DATA_BLOCK "hmiDB"
TITLE = hmiDB
{ S7_Optimized_Access := 'FALSE' }
AUTHOR : JB
VERSION : 0.1
NON_RETAIN
//Contains all the tags that a HMI will need to interact with, sorted in sections. Each cycle, the inputs are read, and the outputs are updated.
   STRUCT
      system : Struct
         general : Struct
            errorPLC { ExternalWritable := 'False'} : Bool;   // Shows error in the PLC
            requestClearFaults : Bool;   // Button input, to clear faults
            systemFault { ExternalWritable := 'False'} : Bool;   // Indicator, to show if fault is present
            faultCount { ExternalWritable := 'False'} : Int;   // Count of how many faults are present
            coolantStatus { ExternalWritable := 'False'} : Bool;   // Indicator, to show if coolant is active
            faultArray { ExternalWritable := 'False'} : Array[0..100] of Bool;
            messageBuffer { ExternalWritable := 'False'} : Array[0..29] of Int;
            bufferIndex { ExternalWritable := 'False'} : Int;
         END_STRUCT;
         ionSource : Struct
            general : Struct
               status : Int;   // Status, enabled=+1, fault=+2
               modeCurrent { ExternalWritable := 'False'} : Int;   // Display field showing source mode
               requestStart : Bool;   // Button input, to start the source
               requestStop : Bool;   // Button input, to stop the source
               requestCondition : Bool;   // Tickbox input
               conditioningPaused { ExternalWritable := 'False'} : Bool;   // Indicator, to show if conditioning has paused
               requestPause : Bool;   // Button input, to pause the source
               requestResume : Bool;   // Button input, to resume the source
               bodyTempC { ExternalWritable := 'False'} : Real;   // Display number, showing source temperature
               bodyTempOkay { ExternalWritable := 'False'} : Bool;   // Indicator, to show if source is cold enough - affects colour of above number
               beamVoltage { ExternalWritable := 'False'} : Real;
               doorStatus : Bool;
            END_STRUCT;
            ioniser : Struct
               status { ExternalWritable := 'False'} : Int;   // Status for ioniser, enabled=+1, fault=+2
               hmiSetpointWEnabled { ExternalWritable := 'False'} : Bool;   // Determines if power setpoint can be written too by HMI
               hmiSetpointWEntry : Real;   // Entry field, to set ioniser power
               hmiSetpointWEntryMin { ExternalWritable := 'False'} : Real;
               hmiSetpointWEntryMax { ExternalWritable := 'False'} : Real;
               readbackW { ExternalWritable := 'False'} : Real;   // Display field, showing ioniser power
               powerRatio : Real;
               filament : Struct
                  status : Int;   // Status, enabled=+1, fault=+2
                  readbackV : Real;
                  readbackA : Real;
                  readbackW : Real;
               END_STRUCT;
               thermionic : Struct
                  status : Int;   // Status, enabled=+1, fault=+2
                  readbackV : Real;
                  readbackA : Real;
                  readbackW : Real;
               END_STRUCT;
            END_STRUCT;
            target : Struct
               status { ExternalWritable := 'False'} : Int;   // Status for target, 0=off/disabled, 1=on/enabled, 2=fault
               hmiSetpointVEnabled { ExternalWritable := 'False'} : Bool;   // Determines if voltage setpoint can be written too by HMI
               hmiSetpointVEntry : Real;   // Entry field, to set target voltage
               hmiSetpointVEntryMin { ExternalWritable := 'False'} : Real;
               hmiSetpointVEntryMax { ExternalWritable := 'False'} : Real;
               readbackV { ExternalWritable := 'False'} : Real;   // Display field, showing target voltage
               readbackA { ExternalWritable := 'False'} : Real;   // Display field, showing target current
               readbackW { ExternalWritable := 'False'} : Real;   // Display field, showing target power
            END_STRUCT;
            extraction : Struct
               status { ExternalWritable := 'False'} : Int;   // Status for extraction, 0=off/disabled, 1=on/enabled, 2=fault
               hmiSetpointVEnabled { ExternalWritable := 'False'} : Bool;   // Determines if extraction setopint can be written too by HMI
               hmiSetpointVEntry : Real;   // Entry field, to set extraction voltage
               hmiSetpointVEntryMin { ExternalWritable := 'False'} : Real;
               hmiSetpointVEntryMax { ExternalWritable := 'False'} : Real;
               readbackV { ExternalWritable := 'False'} : Real;   // Display field, showing extraction voltage
               readbackA { ExternalWritable := 'False'} : Real;   // Display field, showing extraction current
               readbackW { ExternalWritable := 'False'} : Real;   // Display field, showing extraction power
            END_STRUCT;
            cesium : Struct
               status { ExternalWritable := 'False'} : Int;   // Status for cesium, 0=off/disabled, 1=on/enabled, 2=fault
               hmiSetpointCEnabled { ExternalWritable := 'False'} : Bool;   // Determines if temperature setpoint can be written too by HMI
               hmiSetpointCEntry : Real;   // Entry field, to set cesium temperature
               hmiSetpointCEntryMin { ExternalWritable := 'False'} : Real;
               hmiSetpointCEntryMax { ExternalWritable := 'False'} : Real;
               readbackC { ExternalWritable := 'False'} : Real;   // Display field, showing cesium temperature
               heaterOn { ExternalWritable := 'False'} : Bool;   // Indicator, to show if heat is being applied
               coolantOn { ExternalWritable := 'False'} : Bool;   // Indicator, to show if coolant is active
            END_STRUCT;
         END_STRUCT;
         vacuumSystem : Struct
            gauges : Struct
               source : Struct
                  readback_mB : Real;
                  status : Bool;
               END_STRUCT;
               beamline : Struct
                  readback_mB : Real;
                  status : Bool;
               END_STRUCT;
               chamber_UHV_gauge : Struct
                  readback_mB : Bool;
                  status : Bool;
               END_STRUCT;
               chamber_reg_gauge : Struct
                  readback_mB : Real;
                  status : Bool;
               END_STRUCT;
            END_STRUCT;
            pumps : Struct
               roughing { ExternalWritable := 'False'} : Struct
                  source { ExternalWritable := 'False'} : Struct
                     status { ExternalWritable := 'False'} : Bool;
                  END_STRUCT;
                  beamline { ExternalWritable := 'False'} : Struct
                     status { ExternalWritable := 'False'} : Bool;
                  END_STRUCT;
                  loadlock { ExternalWritable := 'False'} : Struct
                     status { ExternalWritable := 'False'} : Bool;
                  END_STRUCT;
               END_STRUCT;
               turbo { ExternalWritable := 'False'} : Struct
                  source_1 { ExternalWritable := 'False'} : Struct
                     status { ExternalWritable := 'False'} : Bool;
                     speed { ExternalWritable := 'False'} : Real;
                     on_hours { ExternalWritable := 'False'} : Real;
                  END_STRUCT;
                  source_2 { ExternalWritable := 'False'} : Struct
                     status { ExternalWritable := 'False'} : Bool;
                     speed { ExternalWritable := 'False'} : Real;
                     on_hours { ExternalWritable := 'False'} : Real;
                  END_STRUCT;
                  beamline { ExternalWritable := 'False'} : Struct
                     status { ExternalWritable := 'False'} : Bool;
                     speed { ExternalWritable := 'False'} : Real;
                     on_hours { ExternalWritable := 'False'} : Real;
                  END_STRUCT;
                  chamber { ExternalWritable := 'False'} : Struct
                     status { ExternalWritable := 'False'} : Bool;
                     speed { ExternalWritable := 'False'} : Real;
                     on_hours { ExternalWritable := 'False'} : Real;
                  END_STRUCT;
                  loadlock { ExternalWritable := 'False'} : Struct
                     status { ExternalWritable := 'False'} : Bool;
                     speed { ExternalWritable := 'False'} : Real;
                     on_hours { ExternalWritable := 'False'} : Real;
                  END_STRUCT;
               END_STRUCT;
               titanium : Struct
                  chamber_1 : Struct
                     on_time_s : Real;
                     off_time_s : Real;
                     nominal_current_A : Real;
                     filament_1 : Struct
                        status : Bool;
                        on_hours : Real;
                        cycles : Int;
                     END_STRUCT;
                  END_STRUCT;
               END_STRUCT;
               ion : Struct
                  chamber_1 : Struct
                     voltage_readback_V : Real;
                     current_readback_A : Real;
                     on_hours : Real;
                  END_STRUCT;
               END_STRUCT;
            END_STRUCT;
            valves : Struct
               gate : Struct
                  "source-beamline" : Struct
                     open : Bool;
                     cycles : Int;
                     requestOpen : Bool;
                  END_STRUCT;
                  "beamline-chamber" : Struct
                     open : Bool;
                     cycles : Int;
                     requestOpen : Bool;
                  END_STRUCT;
                  "chamber-loadlock" : Struct
                     open : Bool;
                     cycles : Int;
                  END_STRUCT;
               END_STRUCT;
               pneumatic : Struct
                  placeholder : Bool;
               END_STRUCT;
            END_STRUCT;
         END_STRUCT;
         beamline : Struct
            magnet : Struct
               status : Int;
               static_active : Bool;
               hmiSetpointAEnabled : Bool;
               hmiSetpointAEntry : Real;
               hmiSetpointAEntryMin : Real;
               hmiSetpointAEntryMax : Real;
               readbackV : Real;
               readbackA : Real;
               outputEnabled : Bool;
               fault : Bool;
            END_STRUCT;
            steerers : Struct
               x : Struct
                  status : Bool;
                  hmiSetpointVEnabled : Bool;
                  hmiSetpointVEntry : Real;
                  hmiSetpointVEntryMin : Real;
                  hmiSetpointVEntryMax : Real;
                  readbackV : Real;
                  readbackA : Real;
                  outputEnabled : Bool;
                  fault : Bool;
               END_STRUCT;
               y : Struct
                  status : Bool;
                  hmiSetpointVEnabled : Bool;
                  hmiSetpointVEntry : Real;
                  hmiSetpointVEntryMin : Real;
                  hmiSetpointVEntryMax : Real;
                  readbackV : Real;
                  readbackA : Real;
                  outputEnabled : Bool;
                  fault : Bool;
               END_STRUCT;
            END_STRUCT;
            einzels : Struct
               lens1 : Struct
                  status : Bool;
                  hmiSetpointVEnabled : Bool;
                  hmiSetpointVEntry : Real;
                  hmiSetpointVEntryMin : Real;
                  hmiSetpointVEntryMax : Real;
                  readbackV : Real;
                  readbackA : Real;
                  outputEnabled : Bool;
                  fault : Bool;
               END_STRUCT;
               lens2 : Struct
                  status : Bool;
                  hmiSetpointVEnabled : Bool;
                  hmiSetpointVEntry : Real;
                  hmiSetpointVEntryMin : Real;
                  hmiSetpointVEntryMax : Real;
                  readbackV : Real;
                  readbackA : Real;
                  outputEnabled : Bool;
                  fault : Bool;
               END_STRUCT;
               lens3 : Struct
                  status : Bool;
                  hmiSetpointVEnabled : Bool;
                  hmiSetpointVEntry : Real;
                  hmiSetpointVEntryMin : Real;
                  hmiSetpointVEntryMax : Real;
                  readbackV : Real;
                  readbackA : Real;
                  outputEnabled : Bool;
                  fault : Bool;
               END_STRUCT;
            END_STRUCT;
            mass_slits : Struct
               left_position : Real;
               right_position : Real;
               gap_width_mm : Real;
               gap_offset_mm : Real;
               bias_voltage : Real;
            END_STRUCT;
            drop_in_cup : Struct
               engaged : Bool;
               requestEngaged : Bool;
               readbackA : Real;
               readbackV : Real;
               hmiSetpointVEntry : Real;
               hmiSetpointVEntryMin : Real;
               hmiSetpointVEntryMax : Real;
            END_STRUCT;
            straight_thru_cup : Struct
               readbackA : Real;
            END_STRUCT;
            massScan : Struct
               requestStart : Bool;
               requestStop : Bool;
               settings : Struct
                  startCurrent : Real;
                  stopCurrent : Real;
                  stepTime : Time;
                  totalSteps : UInt;
                  hystersisWait : Time;
               END_STRUCT;
               feedback : Struct
                  currentStep : UInt;
                  remainingTime_m : UInt;
                  remainingTime_s : UInt;
                  status : Int;   // 0=Idle, 1=Zeroing, 2=Scanning, 99=Error
                  sweepActive : Bool;
                  resultsReady : Bool;
               END_STRUCT;
            END_STRUCT;
         END_STRUCT;
         endstation : Struct
            neutral_trap : Struct
               status : Bool;
               hmiSetpointLeftVEnabled : Bool;
               hmiSetpointLeftVEntry : Real;
               hmiSetpointLeftVEntryMin : Real;
               hmiSetpointLeftVEntryMax : Real;
               readbackLeftV : Real;
               readbackLeftA : Real;
               hmiSetpointRightVEnabled : Bool;
               hmiSetpointRightVEntry : Real;
               hmiSetpointRightVEntryMin : Real;
               hmiSetpointRightVEntryMax : Real;
               readbackRightV : Real;
               readbackRightA : Real;
               fault : Bool;
            END_STRUCT;
            stage : Struct
               motion : Struct
                  status : Int;
                  setpoint_x_mm : Real;
                  setpoint_y_mm : Real;
                  setpoint_z_mm : Real;
                  setpoint_angle_deg : Real;
                  readback_x_mm : Real;
                  readback_y_mm : Real;
                  readback_z_mm : Real;
                  readback_angle_deg : Real;
               END_STRUCT;
               electrical : Struct
                  bias : Real;
                  measured_current_A : Real;
               END_STRUCT;
            END_STRUCT;
            sample : Struct
               status : Int;
               reference_number : Int;
               requested_temp_C : Real;
               measured_temp_C : Real;
               requested_fluence_ions_cm2 : Real;
               measured_fluence_ions_cm2 : Real;
            END_STRUCT;
         END_STRUCT;
      END_STRUCT;
   END_STRUCT;


BEGIN
   system.general.errorPLC := false;
   system.general.requestClearFaults := false;
   system.general.systemFault := false;
   system.general.faultCount := 0;
   system.general.coolantStatus := false;
   system.general.messageBuffer[0] := 0;
   system.general.messageBuffer[1] := 0;
   system.general.messageBuffer[2] := 0;
   system.general.messageBuffer[3] := 0;
   system.general.messageBuffer[4] := 0;
   system.general.messageBuffer[5] := 0;
   system.general.messageBuffer[6] := 0;
   system.general.messageBuffer[7] := 0;
   system.general.messageBuffer[8] := 0;
   system.general.messageBuffer[9] := 0;
   system.general.messageBuffer[10] := 0;
   system.general.messageBuffer[11] := 0;
   system.general.messageBuffer[12] := 0;
   system.general.messageBuffer[13] := 0;
   system.general.messageBuffer[14] := 0;
   system.general.messageBuffer[15] := 0;
   system.general.messageBuffer[16] := 0;
   system.general.messageBuffer[17] := 0;
   system.general.messageBuffer[18] := 0;
   system.general.messageBuffer[19] := 0;
   system.general.messageBuffer[20] := 0;
   system.general.messageBuffer[21] := 0;
   system.general.messageBuffer[22] := 0;
   system.general.messageBuffer[23] := 0;
   system.general.messageBuffer[24] := 0;
   system.general.messageBuffer[25] := 0;
   system.general.messageBuffer[26] := 0;
   system.general.messageBuffer[27] := 0;
   system.general.messageBuffer[28] := 0;
   system.general.messageBuffer[29] := 0;
   system.general.bufferIndex := 0;
   system.ionSource.general.modeCurrent := 0;
   system.ionSource.general.requestStart := false;
   system.ionSource.general.requestStop := false;
   system.ionSource.general.requestCondition := false;
   system.ionSource.general.conditioningPaused := false;
   system.ionSource.general.requestPause := false;
   system.ionSource.general.requestResume := false;
   system.ionSource.general.bodyTempC := 0.0;
   system.ionSource.general.bodyTempOkay := false;
   system.ionSource.general.beamVoltage := 0.0;
   system.ionSource.ioniser.status := 0;
   system.ionSource.ioniser.hmiSetpointWEnabled := false;
   system.ionSource.ioniser.hmiSetpointWEntry := 0.0;
   system.ionSource.ioniser.hmiSetpointWEntryMin := 0.0;
   system.ionSource.ioniser.hmiSetpointWEntryMax := 0.0;
   system.ionSource.ioniser.readbackW := 0.0;
   system.ionSource.target.status := 0;
   system.ionSource.target.hmiSetpointVEnabled := false;
   system.ionSource.target.hmiSetpointVEntry := 0.0;
   system.ionSource.target.hmiSetpointVEntryMin := 0.0;
   system.ionSource.target.hmiSetpointVEntryMax := 0.0;
   system.ionSource.target.readbackV := 0.0;
   system.ionSource.target.readbackA := 0.0;
   system.ionSource.target.readbackW := 0.0;
   system.ionSource.extraction.status := 0;
   system.ionSource.extraction.hmiSetpointVEnabled := false;
   system.ionSource.extraction.hmiSetpointVEntry := 0.0;
   system.ionSource.extraction.hmiSetpointVEntryMin := 0.0;
   system.ionSource.extraction.hmiSetpointVEntryMax := 0.0;
   system.ionSource.extraction.readbackV := 0.0;
   system.ionSource.extraction.readbackA := 0.0;
   system.ionSource.extraction.readbackW := 0.0;
   system.ionSource.cesium.status := 0;
   system.ionSource.cesium.hmiSetpointCEnabled := false;
   system.ionSource.cesium.hmiSetpointCEntry := 40.0;
   system.ionSource.cesium.hmiSetpointCEntryMin := 0.0;
   system.ionSource.cesium.readbackC := 0.0;
   system.ionSource.cesium.heaterOn := false;
   system.ionSource.cesium.coolantOn := false;
   system.beamline.massScan.settings.startCurrent := 0.0;
   system.beamline.massScan.settings.stopCurrent := 10.0;
   system.beamline.massScan.settings.stepTime := T#1S;
   system.beamline.massScan.settings.totalSteps := 30;
   system.beamline.massScan.settings.hystersisWait := T#1000MS;
   system.beamline.massScan.feedback.remainingTime_m := 0;
   system.beamline.massScan.feedback.remainingTime_s := 0;
   system.beamline.massScan.feedback.status := 0;
   system.beamline.massScan.feedback.sweepActive := False;

END_DATA_BLOCK


0.0
0.0
0.0
0.1
0.2
2.0
4.0
6.0
6.0
6.1
6.2
6.3
6.4
6.5
6.6
6.7
7.0
7.1
7.2
7.3
7.4
7.5
7.6
7.7
8.0
8.1
8.2
8.3
8.4
8.5
8.6
8.7
9.0
9.1
9.2
9.3
9.4
9.5
9.6
9.7
10.0
10.1
10.2
10.3
10.4
10.5
10.6
10.7
11.0
11.1
11.2
11.3
11.4
11.5
11.6
11.7
12.0
12.1
12.2
12.3
12.4
12.5
12.6
12.7
13.0
13.1
13.2
13.3
13.4
13.5
13.6
13.7
14.0
14.1
14.2
14.3
14.4
14.5
14.6
14.7
15.0
15.1
15.2
15.3
15.4
15.5
15.6
15.7
16.0
16.1
16.2
16.3
16.4
16.5
16.6
16.7
17.0
17.1
17.2
17.3
17.4
17.5
17.6
17.7
18.0
18.1
18.2
18.3
18.4
20.0
20.0
22.0
24.0
26.0
28.0
30.0
32.0
34.0
36.0
38.0
40.0
42.0
44.0
46.0
48.0
50.0
52.0
54.0
56.0
58.0
60.0
62.0
64.0
66.0
68.0
70.0
72.0
74.0
76.0
78.0
80.0
82.0
82.0
82.0
84.0
86.0
86.1
86.2
86.3
86.4
86.5
88.0
92.0
94.0
98.0
100.0
100.0
102.0
104.0
108.0
112.0
116.0
120.0
124.0
124.0
126.0
130.0
134.0
138.0
138.0
140.0
144.0
148.0
152.0
152.0
154.0
156.0
160.0
164.0
168.0
172.0
176.0
180.0
180.0
182.0
184.0
188.0
192.0
196.0
200.0
204.0
208.0
208.0
210.0
212.0
216.0
220.0
224.0
228.0
228.1
230.0
230.0
230.0
230.0
234.0
236.0
236.0
240.0
242.0
242.0
242.1
244.0
244.0
248.0
250.0
250.0
250.0
250.0
252.0
252.0
254.0
254.0
256.0
256.0
256.0
258.0
262.0
266.0
266.0
268.0
272.0
276.0
276.0
278.0
282.0
286.0
286.0
288.0
292.0
296.0
296.0
298.0
302.0
306.0
306.0
306.0
310.0
314.0
318.0
318.0
320.0
324.0
326.0
326.0
326.0
330.0
334.0
338.0
338.0
338.0
338.0
340.0
342.0
344.0
344.0
346.0
348.0
350.0
350.0
352.0
354.0
354.0
356.0
356.0
356.0
358.0
358.1
360.0
364.0
368.0
372.0
376.0
380.0
380.1
382.0
382.0
382.0
382.1
384.0
388.0
392.0
396.0
400.0
404.0
404.1
406.0
406.0
406.1
408.0
412.0
416.0
420.0
424.0
428.0
428.1
430.0
430.0
430.0
430.1
432.0
436.0
440.0
444.0
448.0
452.0
452.1
454.0
454.0
454.1
456.0
460.0
464.0
468.0
472.0
476.0
476.1
478.0
478.0
478.1
480.0
484.0
488.0
492.0
496.0
500.0
500.1
502.0
502.0
506.0
510.0
514.0
518.0
522.0
522.0
522.1
524.0
528.0
532.0
536.0
540.0
544.0
544.0
548.0
548.0
548.1
550.0
550.0
554.0
558.0
562.0
564.0
568.0
568.0
570.0
572.0
574.0
576.0
576.1
578.0
578.0
578.0
578.1
580.0
584.0
588.0
592.0
596.0
600.0
602.0
606.0
610.0
614.0
618.0
622.0
624.0
624.0
624.0
626.0
630.0
634.0
638.0
642.0
646.0
650.0
654.0
658.0
658.0
662.0
666.0
666.0
668.0
670.0
674.0
678.0
682.0
